# EPICS substitutions: zfmagfldSup/zfmagfld_extra_axis.substitutions
file zfmagfld_cdaq_data.template {
 pattern
    {P, AXIS_INDEX, AXIS, FWDLINK, SCAN}

    {"\$(P)", "3", "EXTRA", "", "1 second"}
}
